KUKA KRL program: A_952154.src, A_952154.dat

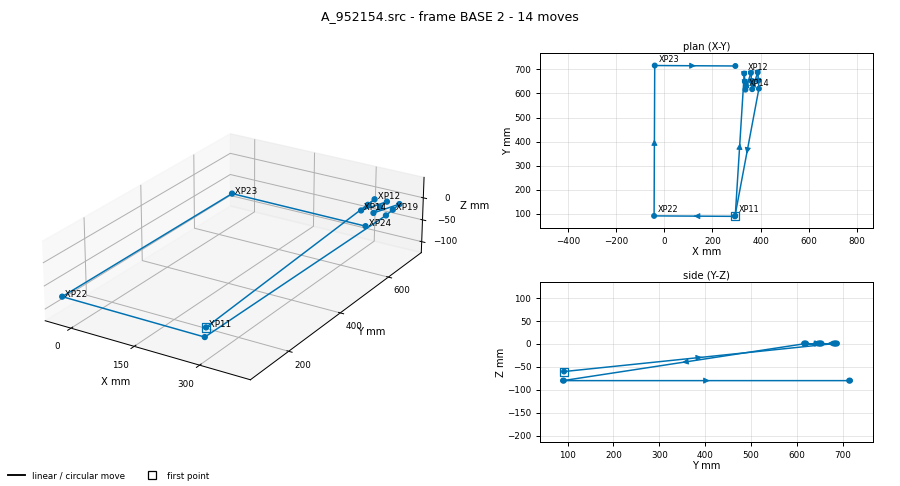
[picture p0: tool path of A_952154.src in frame BASE 2, 14 of 14 moves have a stored position in this frame; points joined in program order, loops and branches not executed]
--- A_952154.src ---
&ACCESS RVO
&REL 641
&PARAM EDITMASK = *
&PARAM TEMPLATE = C:\KRC\Roboter\Template\vorgabe
&PARAM DISKPATH = KRC:\R1\Program\HK
DEF A_952154( )
;FOLD INI;%{PE}
  ;FOLD BASISTECH INI
    GLOBAL INTERRUPT DECL 3 WHEN $STOPMESS==TRUE DO IR_STOPM ( )
    INTERRUPT ON 3
    BAS (#INITMOV,0 )
  ;ENDFOLD (BASISTECH INI)
  ;FOLD USER INI
    ;Make your modifications here

  ;ENDFOLD (USER INI)
;ENDFOLD (INI)



;FOLD PTP P11 Vel=20 % PDAT2 Tool[1]:LASERGUN Base[2]:B_2;%{PE}%R 8.3.48,%MKUKATPBASIS,%CMOVE,%VPTP,%P 1:PTP, 2:P11, 3:, 5:20, 7:PDAT2
$BWDSTART=FALSE
PDAT_ACT=PPDAT2
FDAT_ACT=FP11
BAS(#PTP_PARAMS,20)
PTP XP11
;ENDFOLD
;halt



;FOLD Vision.Calibration_Ini Model:New;%{PE}%MKUKATPUSER


Global_Calib_Model=#New




;ENDFOLD

halt
;FOLD Vision.Calibration_Point Calib_NAME :p12, Calib_NO:1;%{PE}%MKUKATPUSER

HanGao_Calibration_Point(Xp12,1)





;ENDFOLD
;FOLD LIN P12 Vel=.1 m/s CPDAT10 Tool[2]:Work_Tool Base[2]:B_2;%{PE}%R 8.3.48,%MKUKATPBASIS,%CMOVE,%VLIN,%P 1:LIN, 2:P12, 3:, 5:.1, 7:CPDAT10
$BWDSTART=FALSE
LDAT_ACT=LCPDAT10
FDAT_ACT=FP12
BAS(#CP_PARAMS,.1)
LIN XP12
;ENDFOLD

;FOLD Vision.Calibration_Point Calib_NAME :p13, Calib_NO:2;%{PE}%MKUKATPUSER

HanGao_Calibration_Point(Xp13,2)





;ENDFOLD
;FOLD LIN P13 CONT Vel=.1 m/s CPDAT11 Tool[2]:Work_Tool Base[2]:B_2;%{PE}%R 8.3.48,%MKUKATPBASIS,%CMOVE,%VLIN,%P 1:LIN, 2:P13, 3:C_DIS C_DIS, 5:.1, 7:CPDAT11
$BWDSTART=FALSE
LDAT_ACT=LCPDAT11
FDAT_ACT=FP13
BAS(#CP_PARAMS,.1)
LIN XP13 C_DIS C_DIS
;ENDFOLD

;FOLD Vision.Calibration_Point Calib_NAME :p14, Calib_NO:3;%{PE}%MKUKATPUSER

HanGao_Calibration_Point(Xp14,3)





;ENDFOLD
;FOLD LIN P14 Vel=.1 m/s CPDAT12 Tool[2]:Work_Tool Base[2]:B_2;%{PE}%R 8.3.48,%MKUKATPBASIS,%CMOVE,%VLIN,%P 1:LIN, 2:P14, 3:, 5:.1, 7:CPDAT12
$BWDSTART=FALSE
LDAT_ACT=LCPDAT12
FDAT_ACT=FP14
BAS(#CP_PARAMS,.1)
LIN XP14
;ENDFOLD

;FOLD Vision.Calibration_Point Calib_NAME :p15, Calib_NO:4;%{PE}%MKUKATPUSER

HanGao_Calibration_Point(Xp15,4)





;ENDFOLD
;FOLD LIN P15 Vel=.1 m/s CPDAT13 Tool[2]:Work_Tool Base[2]:B_2;%{PE}%R 8.3.48,%MKUKATPBASIS,%CMOVE,%VLIN,%P 1:LIN, 2:P15, 3:, 5:.1, 7:CPDAT13
$BWDSTART=FALSE
LDAT_ACT=LCPDAT13
FDAT_ACT=FP15
BAS(#CP_PARAMS,.1)
LIN XP15
;ENDFOLD

;FOLD Vision.Calibration_Point Calib_NAME :p16, Calib_NO:5;%{PE}%MKUKATPUSER

HanGao_Calibration_Point(Xp16,5)





;ENDFOLD
;FOLD LIN P16 Vel=.1 m/s CPDAT14 Tool[2]:Work_Tool Base[2]:B_2;%{PE}%R 8.3.48,%MKUKATPBASIS,%CMOVE,%VLIN,%P 1:LIN, 2:P16, 3:, 5:.1, 7:CPDAT14
$BWDSTART=FALSE
LDAT_ACT=LCPDAT14
FDAT_ACT=FP16
BAS(#CP_PARAMS,.1)
LIN XP16
;ENDFOLD

;FOLD Vision.Calibration_Point Calib_NAME :p17, Calib_NO:6;%{PE}%MKUKATPUSER

HanGao_Calibration_Point(Xp17,6)





;ENDFOLD
;FOLD LIN P17 Vel=.1 m/s CPDAT15 Tool[2]:Work_Tool Base[2]:B_2;%{PE}%R 8.3.48,%MKUKATPBASIS,%CMOVE,%VLIN,%P 1:LIN, 2:P17, 3:, 5:.1, 7:CPDAT15
$BWDSTART=FALSE
LDAT_ACT=LCPDAT15
FDAT_ACT=FP17
BAS(#CP_PARAMS,.1)
LIN XP17
;ENDFOLD

;FOLD Vision.Calibration_Point Calib_NAME :p18, Calib_NO:7;%{PE}%MKUKATPUSER

HanGao_Calibration_Point(Xp18,7)





;ENDFOLD
;FOLD LIN P18 Vel=.1 m/s CPDAT16 Tool[2]:Work_Tool Base[2]:B_2;%{PE}%R 8.3.48,%MKUKATPBASIS,%CMOVE,%VLIN,%P 1:LIN, 2:P18, 3:, 5:.1, 7:CPDAT16
$BWDSTART=FALSE
LDAT_ACT=LCPDAT16
FDAT_ACT=FP18
BAS(#CP_PARAMS,.1)
LIN XP18
;ENDFOLD

;FOLD Vision.Calibration_Point Calib_NAME :p19, Calib_NO:8;%{PE}%MKUKATPUSER

HanGao_Calibration_Point(Xp19,8)





;ENDFOLD
;FOLD LIN P19 Vel=.1 m/s CPDAT17 Tool[2]:Work_Tool Base[2]:B_2;%{PE}%R 8.3.48,%MKUKATPBASIS,%CMOVE,%VLIN,%P 1:LIN, 2:P19, 3:, 5:.1, 7:CPDAT17
$BWDSTART=FALSE
LDAT_ACT=LCPDAT17
FDAT_ACT=FP19
BAS(#CP_PARAMS,.1)
LIN XP19
;ENDFOLD

;FOLD Vision.Calibration_Point Calib_NAME :p20, Calib_NO:9;%{PE}%MKUKATPUSER

HanGao_Calibration_Point(Xp20,9)





;ENDFOLD
;FOLD LIN P20 Vel=.1 m/s CPDAT19 Tool[2]:Work_Tool Base[2]:B_2;%{PE}%R 8.3.48,%MKUKATPBASIS,%CMOVE,%VLIN,%P 1:LIN, 2:P20, 3:, 5:.1, 7:CPDAT19
$BWDSTART=FALSE
LDAT_ACT=LCPDAT19
FDAT_ACT=FP20
BAS(#CP_PARAMS,.1)
LIN XP20
;ENDFOLD
halt
;loop
;FOLD Vision.Camera_Offset Camera_NAME :P21, Area:45, Work:2;%{PE}%MKUKATPUSER

 HanGao_Camera_Offset(#Calibration ,1,2,XP21)





;ENDFOLD
;FOLD LIN P21 Vel=.1 m/s CPDAT18 Tool[2]:Work_Tool Base[2]:B_2;%{PE}%R 8.3.48,%MKUKATPBASIS,%CMOVE,%VLIN,%P 1:LIN, 2:P21, 3:, 5:.1, 7:CPDAT18
$BWDSTART=FALSE
LDAT_ACT=LCPDAT18
FDAT_ACT=FP21
BAS(#CP_PARAMS,.1)
LIN XP21
;ENDFOLD
;FOLD Vision.Calibration_Send Area:45, Work:2;%{PE}%MKUKATPUSER





EKRL_Calibration_Send("Xml_Vision_Model",1,2)

;ENDFOLD
halt

;FOLD LIN P22 Vel=.1 m/s CPDAT20 Tool[2]:Work_Tool Base[2]:B_2;%{PE}%R 8.3.48,%MKUKATPBASIS,%CMOVE,%VLIN,%P 1:LIN, 2:P22, 3:, 5:.1, 7:CPDAT20
$BWDSTART=FALSE
LDAT_ACT=LCPDAT20
FDAT_ACT=FP22
BAS(#CP_PARAMS,.1)
LIN XP22
;ENDFOLD
;FOLD Vision.Calibration_Send Area:135, Work:2;%{PE}%MKUKATPUSER





EKRL_Calibration_Send("Xml_Vision_Model",2,2)

;ENDFOLD
wait sec 0.1
halt

;FOLD LIN P23 Vel=.1 m/s CPDAT21 Tool[2]:Work_Tool Base[2]:B_2;%{PE}%R 8.3.48,%MKUKATPBASIS,%CMOVE,%VLIN,%P 1:LIN, 2:P23, 3:, 5:.1, 7:CPDAT21
$BWDSTART=FALSE
LDAT_ACT=LCPDAT21
FDAT_ACT=FP23
BAS(#CP_PARAMS,.1)
LIN XP23
;ENDFOLD
;FOLD Vision.Calibration_Send Area:225, Work:2;%{PE}%MKUKATPUSER





EKRL_Calibration_Send("Xml_Vision_Model",3,2)

;ENDFOLD
halt


;FOLD LIN P24 Vel=.1 m/s CPDAT22 Tool[2]:Work_Tool Base[2]:B_2;%{PE}%R 8.3.48,%MKUKATPBASIS,%CMOVE,%VLIN,%P 1:LIN, 2:P24, 3:, 5:.1, 7:CPDAT22
$BWDSTART=FALSE
LDAT_ACT=LCPDAT22
FDAT_ACT=FP24
BAS(#CP_PARAMS,.1)
LIN XP24
;ENDFOLD
;FOLD Vision.Calibration_Send Area:315, Work:2;%{PE}%MKUKATPUSER





EKRL_Calibration_Send("Xml_Vision_Model",4,2)

;ENDFOLD
;endloop
END

--- A_952154.dat ---
&ACCESS RVO
&REL 641
&PARAM EDITMASK = *
&PARAM TEMPLATE = C:\KRC\Roboter\Template\vorgabe
&PARAM DISKPATH = KRC:\R1\Program\HK
DEFDAT  A_952154
;FOLD EXTERNAL DECLARATIONS;%{PE}%MKUKATPBASIS,%CEXT,%VCOMMON,%P
;FOLD BASISTECH EXT;%{PE}%MKUKATPBASIS,%CEXT,%VEXT,%P
EXT  BAS (BAS_COMMAND  :IN,REAL  :IN )
DECL INT SUCCESS
;ENDFOLD (BASISTECH EXT)
;FOLD USER EXT;%{E}%MKUKATPUSER,%CEXT,%VEXT,%P
;Make your modifications here

;ENDFOLD (USER EXT)
;ENDFOLD (EXTERNAL DECLARATIONS)



DECL E6POS XP1={X 962.683960,Y 263.172,Z 756.273499,A 7.43331194,B 44.2248688,C -1.95895112,S 2,T 35,E1 0.0,E2 0.0,E3 0.0,E4 0.0,E5 0.0,E6 0.0}
DECL FDAT FP1={TOOL_NO 1,BASE_NO 0,IPO_FRAME #BASE,POINT2[] " "}
DECL PDAT PPDAT1={VEL 100.000,ACC 100.000,APO_DIST 100.000,APO_MODE #CPTP,GEAR_JERK 100.000,EXAX_IGN 0}
DECL MODULEPARAM_T LAST_TP_PARAMS={PARAMS[] "Kuka.PointName=P10; Kuka.FrameData.base_no=0; Kuka.FrameData.tool_no=1; Kuka.FrameData.ipo_frame=#BASE; Kuka.isglobalpoint=False; Kuka.MoveDataPtpName=PDAT1; Kuka.MovementDataPdat.apo_mode=#CPTP; Kuka.MovementDataPdat.apo_dist=100; Kuka.MovementData.vel=2; Kuka.MovementData.acc=100; Kuka.MovementData.gear_jerk=100; Kuka.MovementData.exax_ign=0; Kuka.VelocityPtp=100; Kuka.BlendingEnabled=False; Kuka.CurrentCDSetIndex=0; Kuka.MoveDataName=CPDAT9; Kuka.MovementData.apo_fac=50; Kuka.MovementData.apo_dist=500; Kuka.MovementData.axis_acc=100; Kuka.MovementData.axis_vel=100; Kuka.MovementData.circ_typ=#BASE; Kuka.MovementData.jerk_fac=50; Kuka.MovementData.ori_typ=#VAR; Kuka.VelocityPath=2               "}
DECL FDAT FS2={TOOL_NO 1,BASE_NO 1,IPO_FRAME #BASE,POINT2[] " ",TQ_STATE FALSE}
DECL LDAT LL2={VEL 0.500000,ACC 1.00000,APO_DIST 10.0000,APO_FAC 50.0000,AXIS_VEL 100.000,AXIS_ACC 100.000,ORI_TYP #VAR,CIRC_TYP #BASE,JERK_FAC 50.0000,GEAR_JERK 50.0000,EXAX_IGN 0}
DECL FDAT FS3={TOOL_NO 1,BASE_NO 1,IPO_FRAME #BASE,POINT2[] " ",TQ_STATE FALSE}
DECL LDAT LL3={VEL 0.500000,ACC 1.00000,APO_DIST 10.0000,APO_FAC 50.0000,AXIS_VEL 100.000,AXIS_ACC 100.000,ORI_TYP #VAR,CIRC_TYP #BASE,JERK_FAC 50.0000,GEAR_JERK 50.0000,EXAX_IGN 0}
DECL FDAT FS5={TOOL_NO 1,BASE_NO 1,IPO_FRAME #BASE,POINT2[] " ",TQ_STATE FALSE}
DECL LDAT LS3={VEL 2.00000,ACC 100.000,APO_DIST 10.0000,APO_FAC 50.0000,AXIS_VEL 100.000,AXIS_ACC 100.000,ORI_TYP #VAR,CIRC_TYP #BASE,JERK_FAC 50.0000,GEAR_JERK 100.000,EXAX_IGN 0}
DECL E6POS POS2={X 0.0,Y 0.0,Z 0.0,A 0.0,B 0.0,C 0.0}
DECL LDAT LL1={VEL 0.400000,ACC 1.00000,APO_DIST 10.0000,APO_FAC 50.0000,AXIS_VEL 100.000,AXIS_ACC 100.000,ORI_TYP #VAR,CIRC_TYP #BASE,JERK_FAC 50.0000,GEAR_JERK 50.0000,EXAX_IGN 0}
DECL E6POS POPM2={X 0.0,Y 0.0,Z 0.0,A 0.0,B 0.0,C 0.0}
DECL E6POS POPE2={X 0.0,Y 0.0,Z 0.0,A 0.0,B 0.0,C 0.0}
DECL FDAT FPE2={TOOL_NO 1,BASE_NO 1,IPO_FRAME #BASE,POINT2[] " ",TQ_STATE FALSE}
DECL LDAT LPM2={VEL 0.0400000,ACC 100.000,APO_DIST 5.00000,APO_FAC 50.0000,AXIS_VEL 100.000,AXIS_ACC 100.000,ORI_TYP #VAR,CIRC_TYP #BASE,JERK_FAC 50.0000,GEAR_JERK 50.0000,EXAX_IGN 0}
DECL E6POS POS3={X 0.0,Y 0.0,Z 0.0,A 0.0,B 0.0,C 0.0}
DECL E6POS POS4={X 0.0,Y 0.0,Z 0.0,A 0.0,B 0.0,C 0.0}
DECL FDAT FS4={TOOL_NO 1,BASE_NO 1,IPO_FRAME #BASE,POINT2[] " ",TQ_STATE FALSE}
DECL LDAT LL4={VEL 0.500000,ACC 1.00000,APO_DIST 10.0000,APO_FAC 50.0000,AXIS_VEL 100.000,AXIS_ACC 100.000,ORI_TYP #VAR,CIRC_TYP #BASE,JERK_FAC 50.0000,GEAR_JERK 50.0000,EXAX_IGN 0}
DECL E6POS POS5={X 0.0,Y 0.0,Z 0.0,A 0.0,B 0.0,C 0.0}
DECL LDAT LL5={VEL 0.01000000,ACC 1.00000,APO_DIST 10.0000,APO_FAC 50.0000,AXIS_VEL 100.000,AXIS_ACC 100.000,ORI_TYP #VAR,CIRC_TYP #BASE,JERK_FAC 50.0000,GEAR_JERK 50.0000,EXAX_IGN 0}
DECL E6POS XP2={X 1765.00,Y -8.79124904E-35,Z 1784.00,A 0.0,B 90.0000,C 2.85383271E-36,S 2,T 34,E1 0.0,E2 0.0,E3 0.0,E4 0.0,E5 0.0,E6 0.0}
DECL FDAT FP2={TOOL_NO 1,BASE_NO 0,IPO_FRAME #BASE,POINT2[] " "}
DECL LDAT LCPDAT1={VEL 2.00000,ACC 100.000,APO_DIST 500.000,APO_FAC 50.0000,AXIS_VEL 100.000,AXIS_ACC 100.000,ORI_TYP #VAR,CIRC_TYP #BASE,JERK_FAC 50.0000,GEAR_JERK 100.000,EXAX_IGN 0}
DECL E6POS XP3={X 1765.00,Y -8.79124904E-35,Z 1784.00,A 0.0,B 90.0000,C 2.85383271E-36,S 2,T 34,E1 0.0,E2 0.0,E3 0.0,E4 0.0,E5 0.0,E6 0.0}
DECL FDAT FP3={TOOL_NO 1,BASE_NO 0,IPO_FRAME #BASE,POINT2[] " "}
DECL LDAT LCPDAT2={VEL 2.00000,ACC 100.000,APO_DIST 500.000,APO_FAC 50.0000,AXIS_VEL 100.000,AXIS_ACC 100.000,ORI_TYP #VAR,CIRC_TYP #BASE,JERK_FAC 50.0000,GEAR_JERK 100.000,EXAX_IGN 0}
DECL E6POS XP4={X 1765.00,Y -8.79124904E-35,Z 1784.00,A 0.0,B 90.0000,C 2.85383271E-36,S 2,T 34,E1 0.0,E2 0.0,E3 0.0,E4 0.0,E5 0.0,E6 0.0}
DECL FDAT FP4={TOOL_NO 1,BASE_NO 0,IPO_FRAME #BASE,POINT2[] " "}
DECL LDAT LCPDAT3={VEL 2.00000,ACC 100.000,APO_DIST 500.000,APO_FAC 50.0000,AXIS_VEL 100.000,AXIS_ACC 100.000,ORI_TYP #VAR,CIRC_TYP #BASE,JERK_FAC 50.0000,GEAR_JERK 100.000,EXAX_IGN 0}
DECL E6POS XP5={X 1765.00,Y -8.79124904E-35,Z 1784.00,A 0.0,B 90.0000,C 2.85383271E-36,S 2,T 34,E1 0.0,E2 0.0,E3 0.0,E4 0.0,E5 0.0,E6 0.0}
DECL FDAT FP5={TOOL_NO 1,BASE_NO 0,IPO_FRAME #BASE,POINT2[] " "}
DECL LDAT LCPDAT4={VEL 2.00000,ACC 100.000,APO_DIST 500.000,APO_FAC 50.0000,AXIS_VEL 100.000,AXIS_ACC 100.000,ORI_TYP #VAR,CIRC_TYP #BASE,JERK_FAC 50.0000,GEAR_JERK 100.000,EXAX_IGN 0}
DECL E6POS XP6={X 1765.00,Y -8.79124904E-35,Z 1784.00,A 0.0,B 90.0000,C 2.85383271E-36,S 2,T 34,E1 0.0,E2 0.0,E3 0.0,E4 0.0,E5 0.0,E6 0.0}
DECL FDAT FP6={TOOL_NO 1,BASE_NO 0,IPO_FRAME #BASE,POINT2[] " "}
DECL LDAT LCPDAT5={VEL 2.00000,ACC 100.000,APO_DIST 500.000,APO_FAC 50.0000,AXIS_VEL 100.000,AXIS_ACC 100.000,ORI_TYP #VAR,CIRC_TYP #BASE,JERK_FAC 50.0000,GEAR_JERK 100.000,EXAX_IGN 0}
DECL E6POS XP7={X 1765.00,Y -8.79124904E-35,Z 1784.00,A 0.0,B 90.0000,C 2.85383271E-36,S 2,T 34,E1 0.0,E2 0.0,E3 0.0,E4 0.0,E5 0.0,E6 0.0}
DECL FDAT FP7={TOOL_NO 1,BASE_NO 0,IPO_FRAME #BASE,POINT2[] " "}
DECL LDAT LCPDAT6={VEL 2.00000,ACC 100.000,APO_DIST 500.000,APO_FAC 50.0000,AXIS_VEL 100.000,AXIS_ACC 100.000,ORI_TYP #VAR,CIRC_TYP #BASE,JERK_FAC 50.0000,GEAR_JERK 100.000,EXAX_IGN 0}
DECL E6POS XP8={X 1765.00,Y -8.79124904E-35,Z 1784.00,A 0.0,B 90.0000,C 2.85383271E-36,S 2,T 34,E1 0.0,E2 0.0,E3 0.0,E4 0.0,E5 0.0,E6 0.0}
DECL FDAT FP8={TOOL_NO 1,BASE_NO 0,IPO_FRAME #BASE,POINT2[] " "}
DECL LDAT LCPDAT7={VEL 2.00000,ACC 100.000,APO_DIST 500.000,APO_FAC 50.0000,AXIS_VEL 100.000,AXIS_ACC 100.000,ORI_TYP #VAR,CIRC_TYP #BASE,JERK_FAC 50.0000,GEAR_JERK 100.000,EXAX_IGN 0}
DECL E6POS XP9={X 1765.00,Y -8.79124904E-35,Z 1784.00,A 0.0,B 90.0000,C 2.85383271E-36,S 2,T 34,E1 0.0,E2 0.0,E3 0.0,E4 0.0,E5 0.0,E6 0.0}
DECL FDAT FP9={TOOL_NO 1,BASE_NO 0,IPO_FRAME #BASE,POINT2[] " "}
DECL LDAT LCPDAT8={VEL 2.00000,ACC 100.000,APO_DIST 500.000,APO_FAC 50.0000,AXIS_VEL 100.000,AXIS_ACC 100.000,ORI_TYP #VAR,CIRC_TYP #BASE,JERK_FAC 50.0000,GEAR_JERK 100.000,EXAX_IGN 0}
DECL E6POS XP10={X 1765.00,Y -8.79124904E-35,Z 1784.00,A 0.0,B 90.0000,C 2.85383271E-36,S 2,T 34,E1 0.0,E2 0.0,E3 0.0,E4 0.0,E5 0.0,E6 0.0}
DECL FDAT FP10={TOOL_NO 1,BASE_NO 0,IPO_FRAME #BASE,POINT2[] " "}
DECL LDAT LCPDAT9={VEL 2.00000,ACC 100.000,APO_DIST 500.000,APO_FAC 50.0000,AXIS_VEL 100.000,AXIS_ACC 100.000,ORI_TYP #VAR,CIRC_TYP #BASE,JERK_FAC 50.0000,GEAR_JERK 100.000,EXAX_IGN 0}
DECL BASIS_SUGG_T LAST_BASIS={POINT1[] "P24                     ",POINT2[] "P24                     ",CP_PARAMS[] "CPDAT22                 ",PTP_PARAMS[] "PDAT3                   ",CONT[] "                        ",CP_VEL[] ".1                      ",PTP_VEL[] "20                      ",SYNC_PARAMS[] "SYNCDAT                 ",SPL_NAME[] "S0                      ",A_PARAMS[] "ADAT0                   "}
DECL E6POS XP11={X 294.592041,Y 92.2328110,Z -60.2262192,A 0.441927105,B -0.0416148715,C -0.0704164654,S 2,T 10,E1 0.0,E2 0.0,E3 0.0,E4 0.0,E5 0.0,E6 0.0}
DECL FDAT FP11={TOOL_NO 1,BASE_NO 2,IPO_FRAME #BASE,POINT2[] " ",TQ_STATE FALSE}
DECL PDAT PPDAT2={VEL 100.000,ACC 100.000,APO_DIST 100.000,GEAR_JERK 50.0000,EXAX_IGN 0}
DECL E6POS XP12={X 331.718597,Y 682.873230,Z 0.925415039,A 0.441951,B -0.0411546156,C -0.104972921,S 2,T 43,E1 0.0,E2 0.0,E3 0.0,E4 0.0,E5 0.0,E6 0.0}
DECL FDAT FP12={TOOL_NO 2,BASE_NO 2,IPO_FRAME #BASE,POINT2[] " ",TQ_STATE FALSE}
DECL LDAT LCPDAT10={VEL 2.00000,ACC 100.000,APO_DIST 100.000,APO_FAC 50.0000,AXIS_VEL 100.000,AXIS_ACC 100.000,ORI_TYP #VAR,CIRC_TYP #BASE,JERK_FAC 50.0000,GEAR_JERK 50.0000,EXAX_IGN 0}
DECL E6POS XP13={X 334.271301,Y 649.548096,Z 0.925419450,A 0.441926658,B -0.0416153371,C -0.0704161823,S 2,T 43,E1 0.0,E2 0.0,E3 0.0,E4 0.0,E5 0.0,E6 0.0}
DECL FDAT FP13={TOOL_NO 2,BASE_NO 2,IPO_FRAME #BASE,POINT2[] " ",TQ_STATE FALSE}
DECL LDAT LCPDAT11={VEL 2.00000,ACC 100.000,APO_DIST 30.0000,APO_FAC 50.0000,AXIS_VEL 100.000,AXIS_ACC 100.000,ORI_TYP #VAR,CIRC_TYP #BASE,JERK_FAC 50.0000,GEAR_JERK 50.0000,EXAX_IGN 0}
DECL E6POS XP14={X 336.839691,Y 615.919922,Z 0.925419450,A 0.441926539,B -0.0416153781,C -0.0704161450,S 2,T 43,E1 0.0,E2 0.0,E3 0.0,E4 0.0,E5 0.0,E6 0.0}
DECL FDAT FP14={TOOL_NO 2,BASE_NO 2,IPO_FRAME #BASE,POINT2[] " ",TQ_STATE FALSE}
DECL LDAT LCPDAT12={VEL 2.00000,ACC 100.000,APO_DIST 100.000,APO_FAC 50.0000,AXIS_VEL 100.000,AXIS_ACC 100.000,ORI_TYP #VAR,CIRC_TYP #BASE,JERK_FAC 50.0000,GEAR_JERK 50.0000,EXAX_IGN 0}
DECL E6POS XP15={X 359.599915,Y 685.269287,Z 0.925419331,A 0.441926450,B -0.0416154228,C -0.0704161301,S 2,T 43,E1 0.0,E2 0.0,E3 0.0,E4 0.0,E5 0.0,E6 0.0}
DECL FDAT FP15={TOOL_NO 2,BASE_NO 2,IPO_FRAME #BASE,POINT2[] " ",TQ_STATE FALSE}
DECL LDAT LCPDAT13={VEL 2.00000,ACC 100.000,APO_DIST 100.000,APO_FAC 50.0000,AXIS_VEL 100.000,AXIS_ACC 100.000,ORI_TYP #VAR,CIRC_TYP #BASE,JERK_FAC 50.0000,GEAR_JERK 50.0000,EXAX_IGN 0}
DECL E6POS XP16={X 362.170807,Y 651.795898,Z 0.925419211,A 0.441926420,B -0.0416154563,C -0.0704161227,S 2,T 43,E1 0.0,E2 0.0,E3 0.0,E4 0.0,E5 0.0,E6 0.0}
DECL FDAT FP16={TOOL_NO 2,BASE_NO 2,IPO_FRAME #BASE,POINT2[] " ",TQ_STATE FALSE}
DECL LDAT LCPDAT14={VEL 2.00000,ACC 100.000,APO_DIST 100.000,APO_FAC 50.0000,AXIS_VEL 100.000,AXIS_ACC 100.000,ORI_TYP #VAR,CIRC_TYP #BASE,JERK_FAC 50.0000,GEAR_JERK 50.0000,EXAX_IGN 0}
DECL E6POS XP17={X 364.744293,Y 617.851624,Z 0.925419152,A 0.441926658,B -0.0416153334,C -0.0704161823,S 2,T 43,E1 0.0,E2 0.0,E3 0.0,E4 0.0,E5 0.0,E6 0.0}
DECL FDAT FP17={TOOL_NO 2,BASE_NO 2,IPO_FRAME #BASE,POINT2[] " ",TQ_STATE FALSE}
DECL LDAT LCPDAT15={VEL 2.00000,ACC 100.000,APO_DIST 100.000,APO_FAC 50.0000,AXIS_VEL 100.000,AXIS_ACC 100.000,ORI_TYP #VAR,CIRC_TYP #BASE,JERK_FAC 50.0000,GEAR_JERK 50.0000,EXAX_IGN 0}
DECL E6POS XP18={X 387.788696,Y 687.522400,Z 0.925419152,A 0.441926330,B -0.0416155085,C -0.0704160854,S 2,T 43,E1 0.0,E2 0.0,E3 0.0,E4 0.0,E5 0.0,E6 0.0}
DECL FDAT FP18={TOOL_NO 2,BASE_NO 2,IPO_FRAME #BASE,POINT2[] " ",TQ_STATE FALSE}
DECL LDAT LCPDAT16={VEL 2.00000,ACC 100.000,APO_DIST 100.000,APO_FAC 50.0000,AXIS_VEL 100.000,AXIS_ACC 100.000,ORI_TYP #VAR,CIRC_TYP #BASE,JERK_FAC 50.0000,GEAR_JERK 50.0000,EXAX_IGN 0}
DECL E6POS XP19={X 390.399475,Y 653.822754,Z 0.925419,A 0.441926628,B -0.0416153409,C -0.0704161748,S 2,T 43,E1 0.0,E2 0.0,E3 0.0,E4 0.0,E5 0.0,E6 0.0}
DECL FDAT FP19={TOOL_NO 2,BASE_NO 2,IPO_FRAME #BASE,POINT2[] " ",TQ_STATE FALSE}
DECL LDAT LCPDAT17={VEL 2.00000,ACC 100.000,APO_DIST 100.000,APO_FAC 50.0000,AXIS_VEL 100.000,AXIS_ACC 100.000,ORI_TYP #VAR,CIRC_TYP #BASE,JERK_FAC 50.0000,GEAR_JERK 50.0000,EXAX_IGN 0}
DECL E6POS XP20={X 392.679688,Y 620.129,Z 0.925418615,A 0.441926599,B -0.0416153707,C -0.0704161674,S 2,T 43,E1 0.0,E2 0.0,E3 0.0,E4 0.0,E5 0.0,E6 0.0}
DECL FDAT FP20={TOOL_NO 2,BASE_NO 2,IPO_FRAME #BASE,POINT2[] " ",TQ_STATE FALSE}
DECL PDAT PPDAT3={VEL 100.000,ACC 100.000,APO_DIST 100.000,GEAR_JERK 50.0000,EXAX_IGN 0}
DECL E6POS XP21={X 293.122131,Y 89.9176636,Z -80.0293961,A 0.441927105,B -0.0416149,C -0.0704163536,S 2,T 10,E1 0.0,E2 0.0,E3 0.0,E4 0.0,E5 0.0,E6 0.0}
DECL FDAT FP21={TOOL_NO 2,BASE_NO 2,IPO_FRAME #BASE,POINT2[] " ",TQ_STATE FALSE}
DECL LDAT LCPDAT18={VEL 2.00000,ACC 100.000,APO_DIST 100.000,APO_FAC 50.0000,AXIS_VEL 100.000,AXIS_ACC 100.000,ORI_TYP #VAR,CIRC_TYP #BASE,JERK_FAC 50.0000,GEAR_JERK 50.0000,EXAX_IGN 0}
DECL LDAT LCPDAT19={VEL 2.00000,ACC 100.000,APO_DIST 100.000,APO_FAC 50.0000,AXIS_VEL 100.000,AXIS_ACC 100.000,ORI_TYP #VAR,CIRC_TYP #BASE,JERK_FAC 50.0000,GEAR_JERK 50.0000,EXAX_IGN 0}
DECL E6POS XP22={X -42.3839874,Y 91.8151550,Z -80.0254822,A 0.441927433,B -0.0416145250,C -0.0704156756,S 2,T 10,E1 0.0,E2 0.0,E3 0.0,E4 0.0,E5 0.0,E6 0.0}
DECL FDAT FP22={TOOL_NO 2,BASE_NO 2,IPO_FRAME #BASE,POINT2[] " ",TQ_STATE FALSE}
DECL LDAT LCPDAT20={VEL 2.00000,ACC 100.000,APO_DIST 100.000,APO_FAC 50.0000,AXIS_VEL 100.000,AXIS_ACC 100.000,ORI_TYP #VAR,CIRC_TYP #BASE,JERK_FAC 50.0000,GEAR_JERK 50.0000,EXAX_IGN 0}
DECL E6POS XP23={X -39.7999954,Y 716.082336,Z -80.0293350,A 0.441926837,B -0.0416151658,C -0.0704162121,S 2,T 43,E1 0.0,E2 0.0,E3 0.0,E4 0.0,E5 0.0,E6 0.0}
DECL FDAT FP23={TOOL_NO 2,BASE_NO 2,IPO_FRAME #BASE,POINT2[] " ",TQ_STATE FALSE}
DECL LDAT LCPDAT21={VEL 2.00000,ACC 100.000,APO_DIST 100.000,APO_FAC 50.0000,AXIS_VEL 100.000,AXIS_ACC 100.000,ORI_TYP #VAR,CIRC_TYP #BASE,JERK_FAC 50.0000,GEAR_JERK 50.0000,EXAX_IGN 0}
DECL E6POS XP24={X 294.984924,Y 714.198059,Z -80.0293350,A 0.441926301,B -0.0416156724,C -0.0704157948,S 2,T 43,E1 0.0,E2 0.0,E3 0.0,E4 0.0,E5 0.0,E6 0.0}
DECL FDAT FP24={TOOL_NO 2,BASE_NO 2,IPO_FRAME #BASE,POINT2[] " ",TQ_STATE FALSE}
DECL LDAT LCPDAT22={VEL 2.00000,ACC 100.000,APO_DIST 100.000,APO_FAC 50.0000,AXIS_VEL 100.000,AXIS_ACC 100.000,ORI_TYP #VAR,CIRC_TYP #BASE,JERK_FAC 50.0000,GEAR_JERK 50.0000,EXAX_IGN 0}
ENDDAT
